FUNCTION_BLOCK LopendeBand
VAR_INPUT
END_VAR
VAR_OUTPUT
END_VAR
VAR
END_VAR

END_FUNCTION_BLOCK

(* stored: Version 1.1.0.1
   POU LopendeBand: Id {af1489a2-4b96-41ec-9023-dbc3371340a0}, SpecialFunc None *)
